// TIA Portal V16 export
// export: Created 2021-04-13T11:10:15.4657649Z, ExportSetting WithDefaults, DisplayName Totally Integrated Automation Portal, DisplayVersion V16, DisplayName TIA Portal Version Control Interface, DisplayVersion V16, DisplayName TIA Portal Openness, DisplayVersion V16, DisplayName STEP 7 Professional, DisplayVersion V16, DisplayName STEP 7 Safety, DisplayVersion V16, DisplayName WinCC Unified SCADA Engineering System, DisplayVersion V16
FUNCTION "IOtoDB" : Void   // FC1, LAD
{ S7_Optimized_Access := 'TRUE' }
VERSION : 0.1
// stored: AutoNumber false, IsIECCheckEnabled false, SetENOAutomatically false, UDAEnableTagReadback false
BEGIN

REGION Network 1: Передаем входа
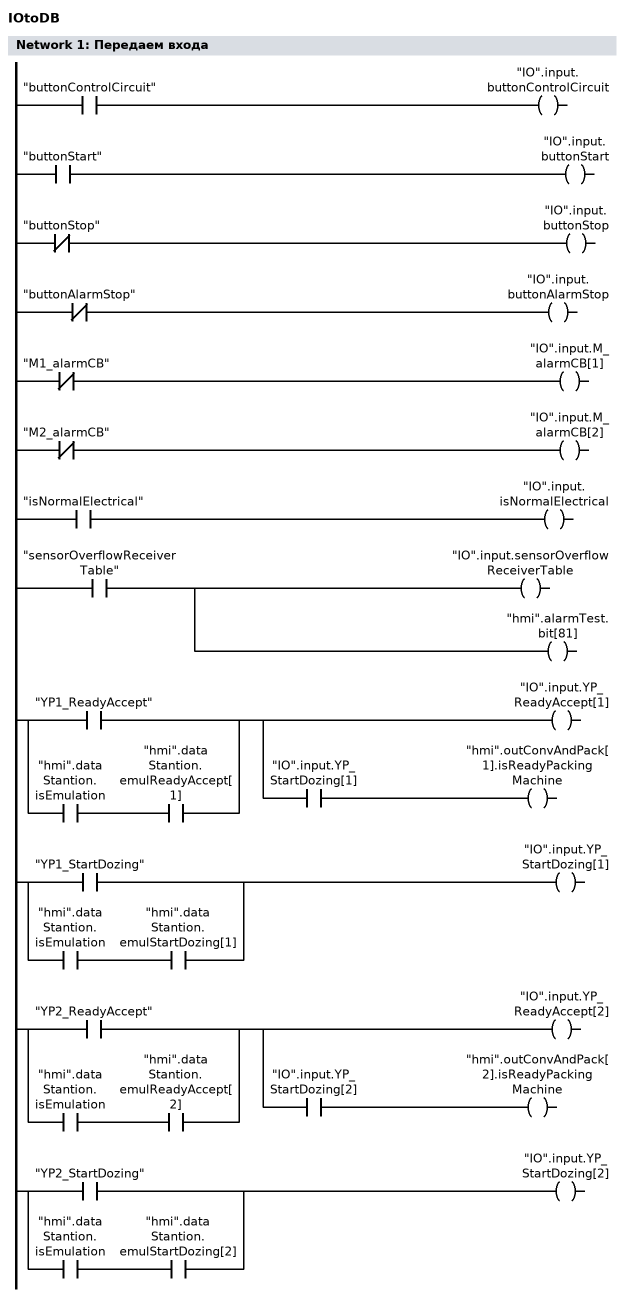
   RUNG wire#powerrail
      Contact( "buttonControlCircuit" )
      Coil( "IO".input.buttonControlCircuit )
   END_RUNG
   RUNG wire#powerrail
      Contact( "buttonStart" )
      Coil( "IO".input.buttonStart )
   END_RUNG
   RUNG wire#powerrail
      I_Contact( "buttonStop" )
      Coil( "IO".input.buttonStop )
   END_RUNG
   RUNG wire#powerrail
      I_Contact( "buttonAlarmStop" )
      Coil( "IO".input.buttonAlarmStop )
   END_RUNG
   RUNG wire#powerrail
      I_Contact( "M1_alarmCB" )
      Coil( "IO".input.M_alarmCB[1] )
   END_RUNG
   RUNG wire#powerrail
      I_Contact( "M2_alarmCB" )
      Coil( "IO".input.M_alarmCB[2] )
   END_RUNG
   RUNG wire#powerrail
      Contact( "isNormalElectrical" )
      Coil( "IO".input.isNormalElectrical )
   END_RUNG
   RUNG wire#powerrail
      Contact( "sensorOverflowReceiverTable" )
      wire#w1
      Coil( "IO".input.sensorOverflowReceiverTable )
   END_RUNG
   RUNG wire#w1
      Coil( "hmi".alarmTest.bit[81] )
   END_RUNG
   RUNG wire#powerrail
      Contact( "YP1_ReadyAccept" )
      wire#w2
      Coil( "IO".input.YP_ReadyAccept[1] )
   END_RUNG
   RUNG wire#powerrail
      Contact( "hmi".dataStantion.isEmulation )
      Contact( "hmi".dataStantion.emulReadyAccept[1] )
   END_RUNG wire#w2
   RUNG wire#w2
      Contact( "IO".input.YP_StartDozing[1] )
      Coil( "hmi".outConvAndPack[1].isReadyPackingMachine )
   END_RUNG
   RUNG wire#powerrail
      Contact( "YP1_StartDozing" )
      wire#w3
      Coil( "IO".input.YP_StartDozing[1] )
   END_RUNG
   RUNG wire#powerrail
      Contact( "hmi".dataStantion.isEmulation )
      Contact( "hmi".dataStantion.emulStartDozing[1] )
   END_RUNG wire#w3
   RUNG wire#powerrail
      Contact( "YP2_ReadyAccept" )
      wire#w4
      Coil( "IO".input.YP_ReadyAccept[2] )
   END_RUNG
   RUNG wire#powerrail
      Contact( "hmi".dataStantion.isEmulation )
      Contact( "hmi".dataStantion.emulReadyAccept[2] )
   END_RUNG wire#w4
   RUNG wire#w4
      Contact( "IO".input.YP_StartDozing[2] )
      Coil( "hmi".outConvAndPack[2].isReadyPackingMachine )
   END_RUNG
   RUNG wire#powerrail
      Contact( "YP2_StartDozing" )
      wire#w5
      Coil( "IO".input.YP_StartDozing[2] )
   END_RUNG
   RUNG wire#powerrail
      Contact( "hmi".dataStantion.isEmulation )
      Contact( "hmi".dataStantion.emulStartDozing[2] )
   END_RUNG wire#w5
   // the same network as SCL:
   "IO".input.buttonControlCircuit := "buttonControlCircuit";
   "IO".input.buttonStart := "buttonStart";
   "IO".input.buttonStop := NOT "buttonStop";
   "IO".input.buttonAlarmStop := NOT "buttonAlarmStop";
   "IO".input.M_alarmCB[1] := NOT "M1_alarmCB";
   "IO".input.M_alarmCB[2] := NOT "M2_alarmCB";
   "IO".input.isNormalElectrical := "isNormalElectrical";
   "IO".input.sensorOverflowReceiverTable := "sensorOverflowReceiverTable";
   "hmi".alarmTest.bit[81] := "sensorOverflowReceiverTable";
   "IO".input.YP_ReadyAccept[1] := "YP1_ReadyAccept" OR ("hmi".dataStantion.isEmulation AND "hmi".dataStantion.emulReadyAccept[1]);
   "hmi".outConvAndPack[1].isReadyPackingMachine := ("YP1_ReadyAccept" OR ("hmi".dataStantion.isEmulation AND "hmi".dataStantion.emulReadyAccept[1])) AND "IO".input.YP_StartDozing[1];
   "IO".input.YP_StartDozing[1] := "YP1_StartDozing" OR ("hmi".dataStantion.isEmulation AND "hmi".dataStantion.emulStartDozing[1]);
   "IO".input.YP_ReadyAccept[2] := "YP2_ReadyAccept" OR ("hmi".dataStantion.isEmulation AND "hmi".dataStantion.emulReadyAccept[2]);
   "hmi".outConvAndPack[2].isReadyPackingMachine := ("YP2_ReadyAccept" OR ("hmi".dataStantion.isEmulation AND "hmi".dataStantion.emulReadyAccept[2])) AND "IO".input.YP_StartDozing[2];
   "IO".input.YP_StartDozing[2] := "YP2_StartDozing" OR ("hmi".dataStantion.isEmulation AND "hmi".dataStantion.emulStartDozing[2]);
END_REGION
END_FUNCTION
